Omron CX-Programmer project NewProject (CX-Programmer 9.75)

# PLC NewPLC1: CJ1M CPU11

## Global symbols (name address type ; comment)
20.00 BOOL  ; Start & Reset
20.01 BOOL  ; Kiln Consent
20.02 BOOL  ; Power OK
20.03 BOOL  ; Manual/Automatic Selector
20.04 BOOL  ; FT Enter Kiln
20.06 BOOL  ; FT Before Barrier
20.07 BOOL  ; FT Row Complete in Belts
20.08 BOOL  ; FT Row In Position
20.09 BOOL  ; FT Step-to-Step
20.10 BOOL  ; Belt Up Sensor
20.11 BOOL  ; Belt Down Sensor
20.12 BOOL  ; FT Wide Largest Row
20.13 BOOL  ; Spare
20.14 BOOL  ; Spare
20.15 BOOL  ; Spare
21.00 BOOL  ; Manual Up/Down Up
21.01 BOOL  ; Manual Up/Down Down
21.02 BOOL  ; Manual Step-To-Step Belts
21.03 BOOL  ; Manual Rollers Under Belts
21.04 BOOL  ; Manual Roller Before Barrier
21.05 BOOL  ; Manual Roller After Barrier
21.06 BOOL  ; Manual Barier Up/Down
21.07 BOOL  ; Manual Prepare Row Valve
21.08 BOOL  ; Spare
21.09 BOOL  ; Spare
21.10 BOOL  ; Spare
21.11 BOOL  ; Spare
21.12 BOOL  ; Spare
21.13 BOOL  ; Spare
21.14 BOOL  ; Spare
21.15 BOOL  ; Spare
30.00 BOOL  ; Enter Kiln Roller
30.01 BOOL  ; Barrier Valve
30.02 BOOL  ; Roller Under Barrier
30.03 BOOL  ; Roller Under Belts
30.04 BOOL  ; Up/Down Belts
30.05 BOOL  ; Up/Down Valve
30.06 BOOL  ; Preapare Row Valve
30.07 BOOL  ; Automatic Run Lamp
30.08 BOOL  ; Spare
30.09 BOOL  ; Spare
30.10 BOOL  ; Enter Kiln Roller (Slow Speed)
30.11 BOOL  ; Roller Under Barrier (Slow Speed)
30.12 BOOL  ; Sarin
30.13 BOOL  ; Sarin
30.14 BOOL  ; Unloaing Machine Consent
30.15 BOOL  ; Unloaing Machine Consent
40.00 BOOL  ; Automatic In progress
40.01 BOOL  ; Automatic Run OK
41.00 BOOL  ; Start Sequence
42.00 BOOL  ; OK Run EnterKiln Rollers
43.00 BOOL  ; Ok Run Roller Under Barrier
50.00 BOOL  ; Existence Alarm
60 CHANNEL  ; Alarms Word
70.00 BOOL  ; Start Sarin
C0001 BOOL  ; Start Fast Speed Enter Kiln Rollers Time
C0002 BOOL  ; Time Slow Speed Roller Under Barrier
C0003 BOOL  ; Stay Barrier Down Down
D100 CHANNEL  ; Start Fast Speed Enter Kiln Rollers Time
D101 CHANNEL  ; Data Time Slow Speed Roller Under Barrier
D102 CHANNEL  ; Time Barrier Stay Down
T0000 BOOL  ; Time Sarin In Start
T0001 BOOL  ; Time FT Enter Kiln Engage
T0002 BOOL  ; Time FT Enter Kiln Disengage
T0003 BOOL  ; FT Large Row Engage
T0004 BOOL  ; FT Large Row Disengage
T0005 BOOL  ; Time Restart Enter Kiln Roller
T0006 BOOL  ; Time FT Befor Brrier Engage
T0007 BOOL  ; Time FT Befor Brrier Disengage
W10.00 BOOL  ; Barrier Valve Up
W11.00 BOOL  ; Up Barrier
W11.01 BOOL  ; Down Barrier

## Program NewProgram1 (cyclic task 0)
; This Program Designed By Eng: Mahmoud Shaban Ahmed

### Section Inputs

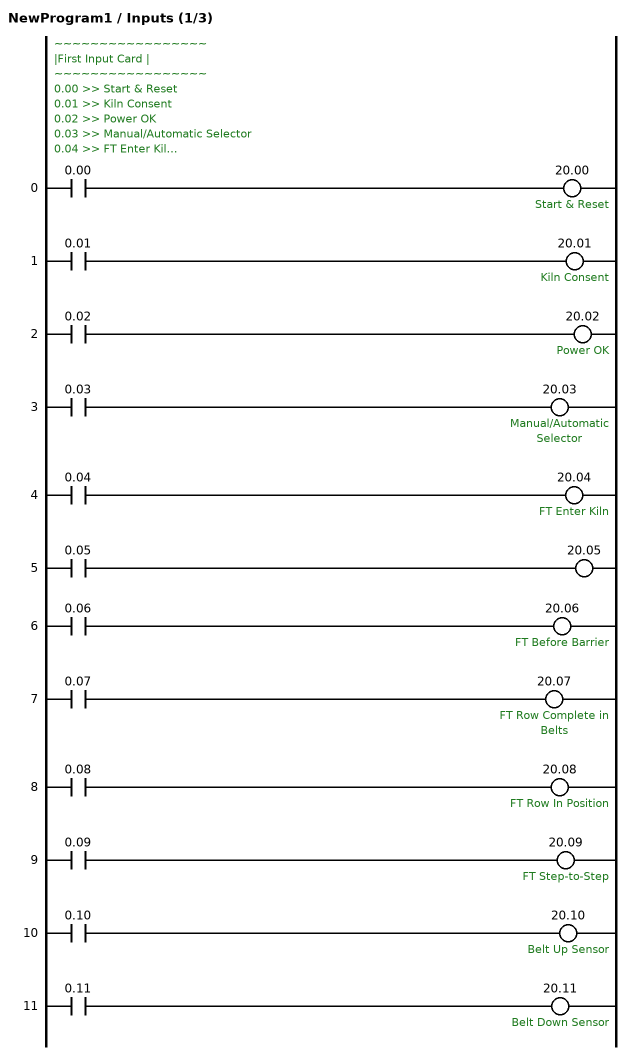
; rung 0: ~~~~~~~~~~~~~~~~~ / |First Input Card | / ~~~~~~~~~~~~~~~~~ / 0.00 >> Start & Reset / 0.01 >> Kiln Consent / 0.02 >> Power OK / 0.03 >> Manual/Automatic Selector / 0.04 >> FT Enter Kiln / 0.05 >> / 0.06 >> FT Before Barrier / 0.07 >> FT Row Complete in Belts / 0.08 >> FT Row In Position / 0.09 >> FT Step-to-Step / 0.10 >> Belt Up Sensor / 0.11 >> Belt Down Sensor / 0.12 >> FT Wide Largest Row / 0.13 >>Spare / 0.14 >>Spare / 0.15 >>Spare / >>>>>>>>>>>>>>>>>>>>>>>>>>>>>>>>>>>>>>>>>>>>>>>>>>>>>>>>>>>>>>>>>>>>>>>>>>>>>>>>>>>>>>>>>>>>>>>>>>>>>>>>>>>>>>>
LD 0.00
OUT 20.00  ; Start & Reset
; rung 1
LD 0.01
OUT 20.01  ; Kiln Consent
; rung 2
LD 0.02
OUT 20.02  ; Power OK
; rung 3
LD 0.03
OUT 20.03  ; Manual/Automatic Selector
; rung 4
LD 0.04
OUT 20.04  ; FT Enter Kiln
; rung 5
LD 0.05
OUT 20.05
; rung 6
LD 0.06
OUT 20.06  ; FT Before Barrier
; rung 7
LD 0.07
OUT 20.07  ; FT Row Complete in Belts
; rung 8
LD 0.08
OUT 20.08  ; FT Row In Position
; rung 9
LD 0.09
OUT 20.09  ; FT Step-to-Step
; rung 10
LD 0.10
OUT 20.10  ; Belt Up Sensor
; rung 11
LD 0.11
OUT 20.11  ; Belt Down Sensor

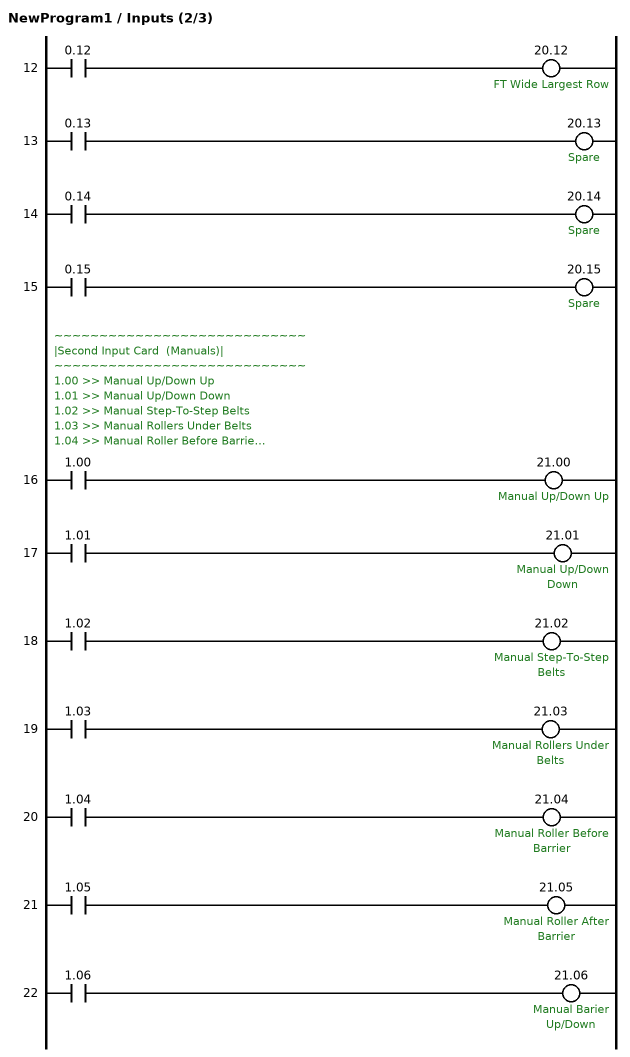
; rung 12
LD 0.12
OUT 20.12  ; FT Wide Largest Row
; rung 13
LD 0.13
OUT 20.13  ; Spare
; rung 14
LD 0.14
OUT 20.14  ; Spare
; rung 15
LD 0.15
OUT 20.15  ; Spare
; rung 16: ~~~~~~~~~~~~~~~~~~~~~~~~~~~~ / |Second Input Card  (Manuals)| / ~~~~~~~~~~~~~~~~~~~~~~~~~~~~ / 1.00 >> Manual Up/Down Up / 1.01 >> Manual Up/Down Down / 1.02 >> Manual Step-To-Step Belts / 1.03 >> Manual Rollers Under Belts / 1.04 >> Manual Roller Before Barrier / 1.05 >> Manual Roller After Barrier / 1.06 >> Manual Barier Up/Down / 1.07 >> Manual Prepare Row Valve / 1.08 >> Spare / 1.09 >> Spare / 1.10 >> Spare / 1.11 >> Spare / 1.12 >> Spare / 1.13 >> Spare / 1.14 >> Spare / 1.15 >> Spare / >>>>>>>>>>>>>>>>>>>>>>>>>>>>>>>>>>>>>>>>>>>>>>>>>>>>>>>>>>>>>>>>>>>>>>>>>>>>>>>>>>>>>>>>>>>>>>>>>>>>>>>>>>>>>>>
LD 1.00
OUT 21.00  ; Manual Up/Down Up
; rung 17
LD 1.01
OUT 21.01  ; Manual Up/Down Down
; rung 18
LD 1.02
OUT 21.02  ; Manual Step-To-Step Belts
; rung 19
LD 1.03
OUT 21.03  ; Manual Rollers Under Belts
; rung 20
LD 1.04
OUT 21.04  ; Manual Roller Before Barrier
; rung 21
LD 1.05
OUT 21.05  ; Manual Roller After Barrier
; rung 22
LD 1.06
OUT 21.06  ; Manual Barier Up/Down

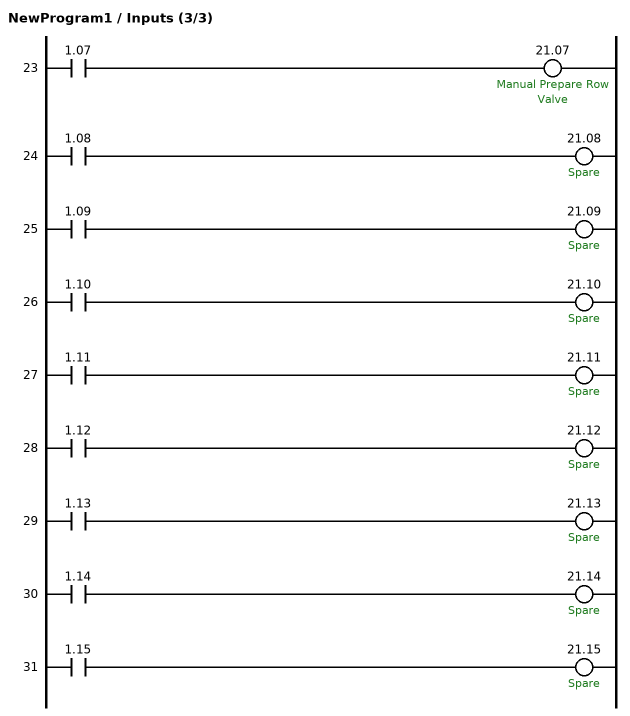
; rung 23
LD 1.07
OUT 21.07  ; Manual Prepare Row Valve
; rung 24
LD 1.08
OUT 21.08  ; Spare
; rung 25
LD 1.09
OUT 21.09  ; Spare
; rung 26
LD 1.10
OUT 21.10  ; Spare
; rung 27
LD 1.11
OUT 21.11  ; Spare
; rung 28
LD 1.12
OUT 21.12  ; Spare
; rung 29
LD 1.13
OUT 21.13  ; Spare
; rung 30
LD 1.14
OUT 21.14  ; Spare
; rung 31
LD 1.15
OUT 21.15  ; Spare

### Section Main

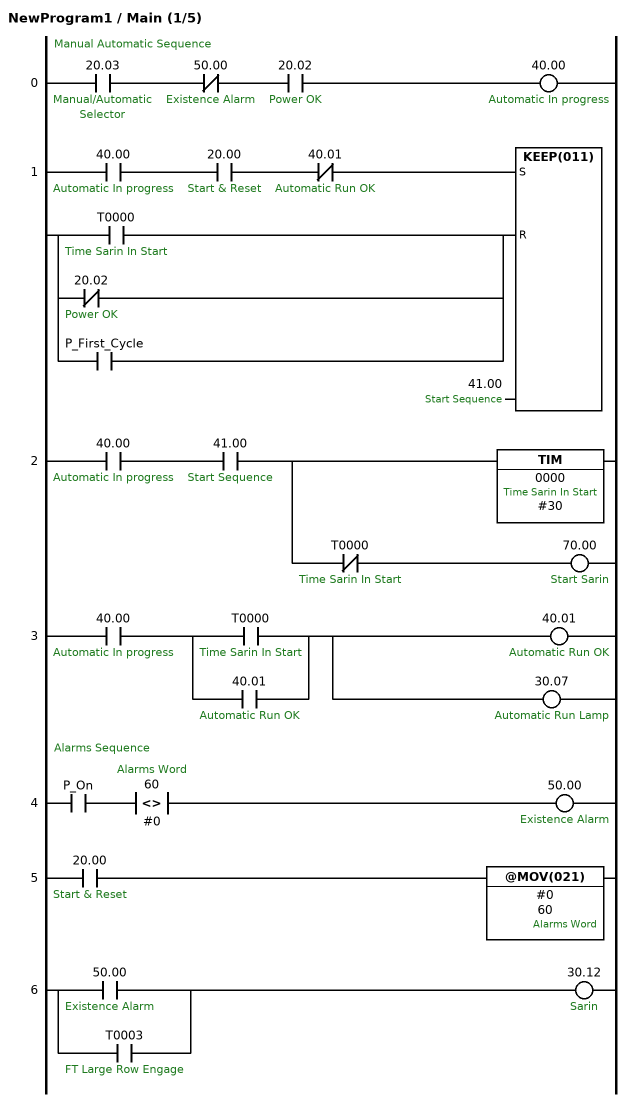
; rung 0: Manual Automatic Sequence
LD 20.03  ; Manual/Automatic Selector
ANDNOT 50.00  ; Existence Alarm
AND 20.02  ; Power OK
OUT 40.00  ; Automatic In progress
; rung 1
LD 40.00  ; Automatic In progress
AND 20.00  ; Start & Reset
ANDNOT 40.01  ; Automatic Run OK
LD T0000  ; Time Sarin In Start
ORNOT 20.02  ; Power OK
OR P_First_Cycle
KEEP(011) 41.00  ; Start Sequence
; rung 2
LD 40.00  ; Automatic In progress
AND 41.00  ; Start Sequence
TIM 0000 #30  ; Time Sarin In Start
ANDNOT T0000  ; Time Sarin In Start
OUT 70.00  ; Start Sarin
; rung 3
LD 40.00  ; Automatic In progress
LD T0000  ; Time Sarin In Start
OR 40.01  ; Automatic Run OK
ANDLD
OUT 40.01  ; Automatic Run OK
OUT 30.07  ; Automatic Run Lamp
; rung 4: Alarms Sequence
LD P_On
AND<>(305) 60 #0  ; Alarms Word
OUT 50.00  ; Existence Alarm
; rung 5
LD 20.00  ; Start & Reset
@MOV(021) #0 60  ; Alarms Word
; rung 6
LD 50.00  ; Existence Alarm
OR T0003  ; FT Large Row Engage
OUT 30.12  ; Sarin

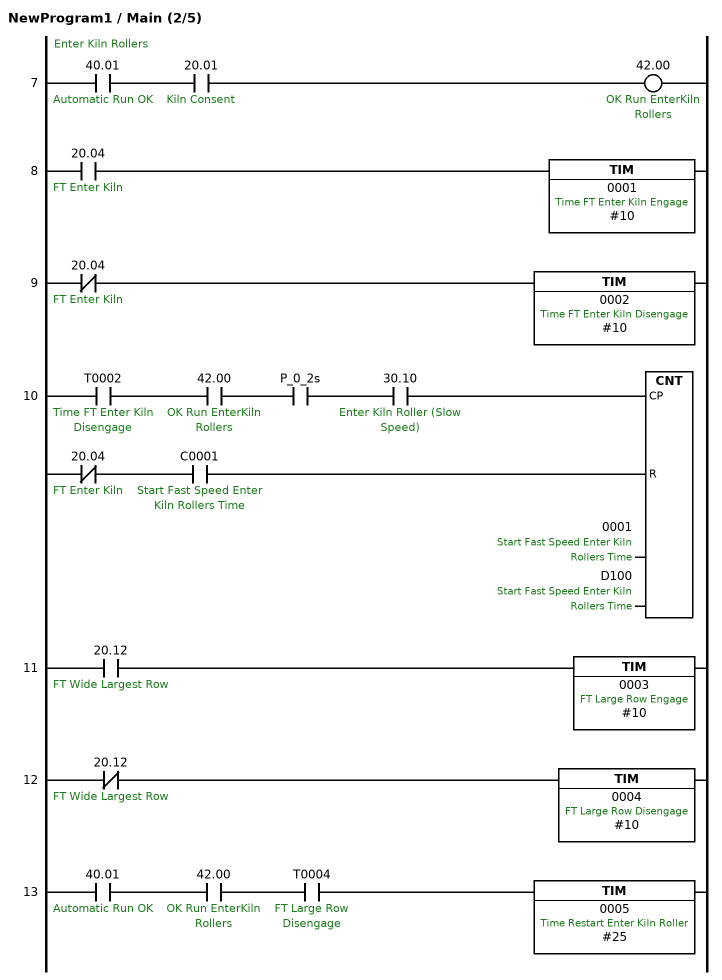
; rung 7: Enter Kiln Rollers
LD 40.01  ; Automatic Run OK
AND 20.01  ; Kiln Consent
OUT 42.00  ; OK Run EnterKiln Rollers
; rung 8
LD 20.04  ; FT Enter Kiln
TIM 0001 #10  ; Time FT Enter Kiln Engage
; rung 9
LDNOT 20.04  ; FT Enter Kiln
TIM 0002 #10  ; Time FT Enter Kiln Disengage
; rung 10
LD T0002  ; Time FT Enter Kiln Disengage
AND 42.00  ; OK Run EnterKiln Rollers
AND P_0_2s
AND 30.10  ; Enter Kiln Roller (Slow Speed)
LDNOT 20.04  ; FT Enter Kiln
AND C0001  ; Start Fast Speed Enter Kiln Rollers Time
CNT 0001 D100  ; Start Fast Speed Enter Kiln Rollers Time
; rung 11
LD 20.12  ; FT Wide Largest Row
TIM 0003 #10  ; FT Large Row Engage
; rung 12
LDNOT 20.12  ; FT Wide Largest Row
TIM 0004 #10  ; FT Large Row Disengage
; rung 13
LD 40.01  ; Automatic Run OK
AND 42.00  ; OK Run EnterKiln Rollers
AND T0004  ; FT Large Row Disengage
TIM 0005 #25  ; Time Restart Enter Kiln Roller

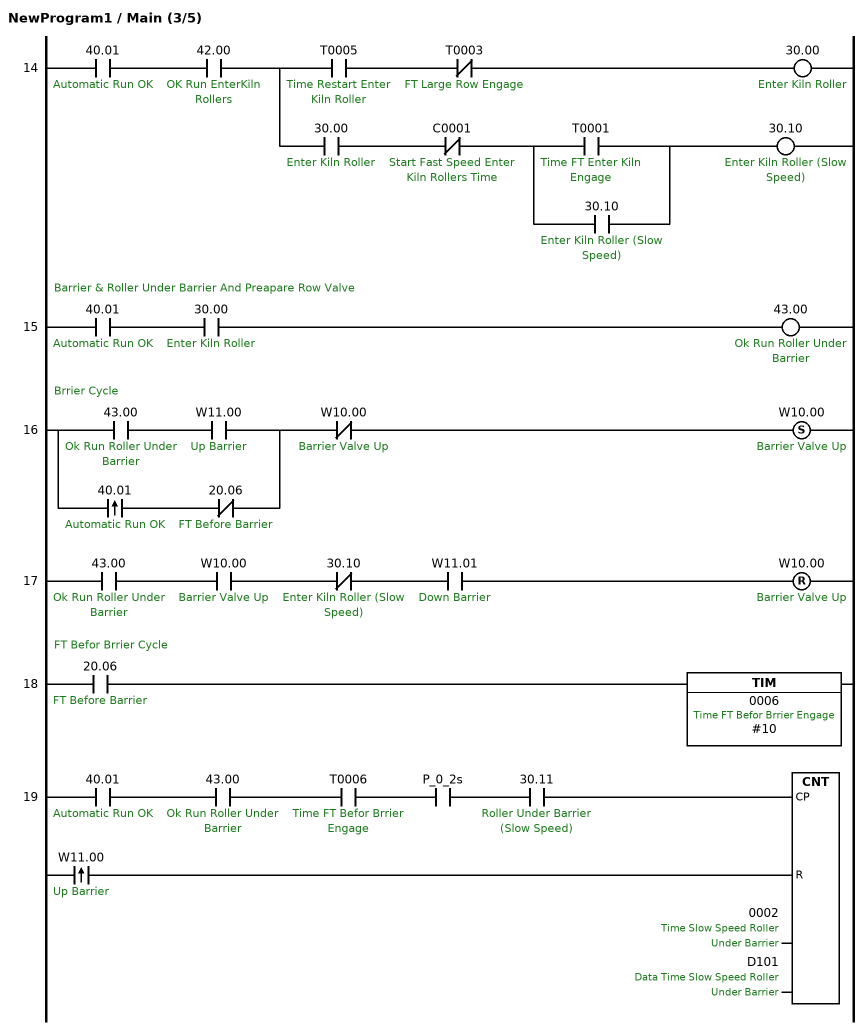
; rung 14
LD 40.01  ; Automatic Run OK
AND 42.00  ; OK Run EnterKiln Rollers
OUT TR0
AND T0005  ; Time Restart Enter Kiln Roller
ANDNOT T0003  ; FT Large Row Engage
OUT 30.00  ; Enter Kiln Roller
LD TR0
AND 30.00  ; Enter Kiln Roller
ANDNOT C0001  ; Start Fast Speed Enter Kiln Rollers Time
LD T0001  ; Time FT Enter Kiln Engage
OR 30.10  ; Enter Kiln Roller (Slow Speed)
ANDLD
OUT 30.10  ; Enter Kiln Roller (Slow Speed)
; rung 15: Barrier & Roller Under Barrier And Preapare Row Valve
LD 40.01  ; Automatic Run OK
AND 30.00  ; Enter Kiln Roller
OUT 43.00  ; Ok Run Roller Under Barrier
; rung 16: Brrier Cycle
LD 43.00  ; Ok Run Roller Under Barrier
AND W11.00  ; Up Barrier
@LD 40.01  ; Automatic Run OK
ANDNOT 20.06  ; FT Before Barrier
ORLD
ANDNOT W10.00  ; Barrier Valve Up
SET W10.00  ; Barrier Valve Up
; rung 17
LD 43.00  ; Ok Run Roller Under Barrier
AND W10.00  ; Barrier Valve Up
ANDNOT 30.10  ; Enter Kiln Roller (Slow Speed)
AND W11.01  ; Down Barrier
RSET W10.00  ; Barrier Valve Up
; rung 18: FT Befor Brrier Cycle
LD 20.06  ; FT Before Barrier
TIM 0006 #10  ; Time FT Befor Brrier Engage
; rung 19
LD 40.01  ; Automatic Run OK
AND 43.00  ; Ok Run Roller Under Barrier
AND T0006  ; Time FT Befor Brrier Engage
AND P_0_2s
AND 30.11  ; Roller Under Barrier (Slow Speed)
@LD W11.00  ; Up Barrier
CNT 0002 D101  ; Data Time Slow Speed Roller Under Barrier, Time Slow Speed Roller Under Barrier

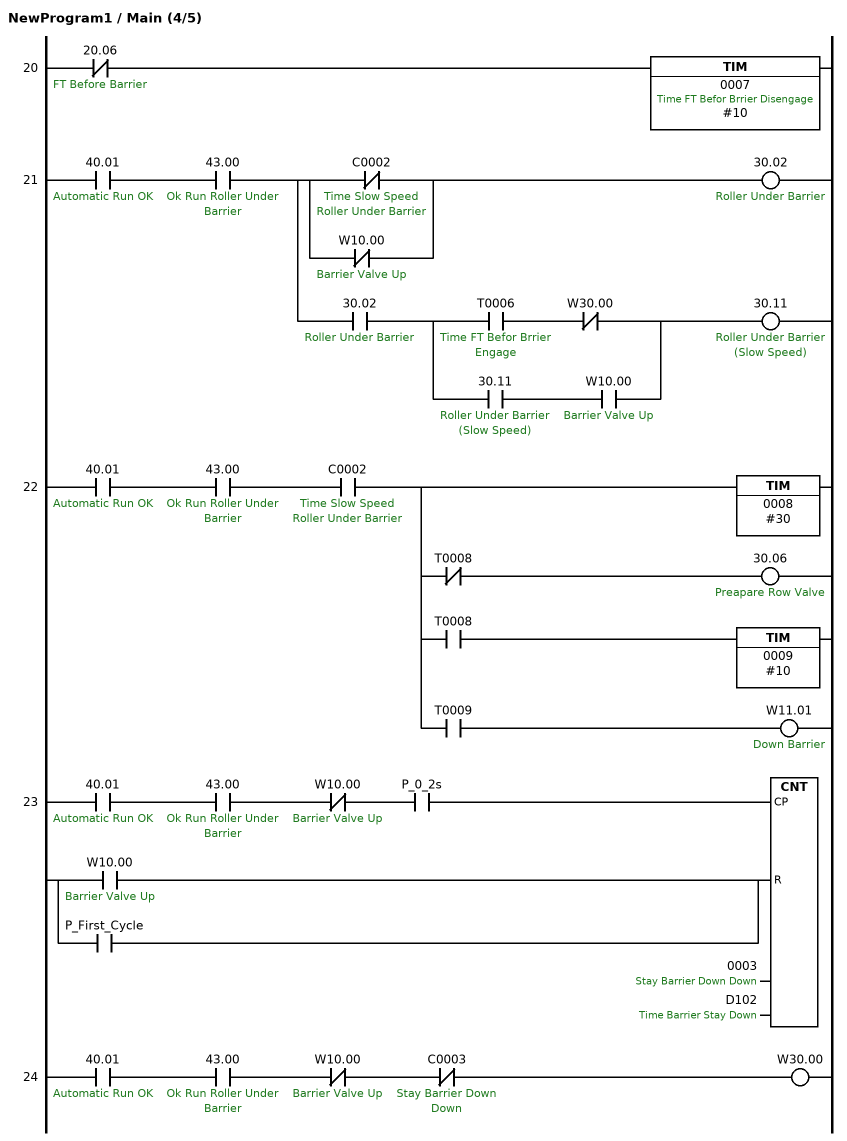
; rung 20
LDNOT 20.06  ; FT Before Barrier
TIM 0007 #10  ; Time FT Befor Brrier Disengage
; rung 21
LD 40.01  ; Automatic Run OK
AND 43.00  ; Ok Run Roller Under Barrier
OUT TR0
LDNOT C0002  ; Time Slow Speed Roller Under Barrier
ORNOT W10.00  ; Barrier Valve Up
ANDLD
OUT 30.02  ; Roller Under Barrier
LD TR0
AND 30.02  ; Roller Under Barrier
LD T0006  ; Time FT Befor Brrier Engage
ANDNOT W30.00
LD 30.11  ; Roller Under Barrier (Slow Speed)
AND W10.00  ; Barrier Valve Up
ORLD
ANDLD
OUT 30.11  ; Roller Under Barrier (Slow Speed)
; rung 22
LD 40.01  ; Automatic Run OK
AND 43.00  ; Ok Run Roller Under Barrier
AND C0002  ; Time Slow Speed Roller Under Barrier
OUT TR0
TIM 0008 #30
ANDNOT T0008
OUT 30.06  ; Preapare Row Valve
LD TR0
AND T0008
TIM 0009 #10
LD TR0
AND T0009
OUT W11.01  ; Down Barrier
; rung 23
LD 40.01  ; Automatic Run OK
AND 43.00  ; Ok Run Roller Under Barrier
ANDNOT W10.00  ; Barrier Valve Up
AND P_0_2s
LD W10.00  ; Barrier Valve Up
OR P_First_Cycle
CNT 0003 D102  ; Time Barrier Stay Down, Stay Barrier Down Down
; rung 24
LD 40.01  ; Automatic Run OK
AND 43.00  ; Ok Run Roller Under Barrier
ANDNOT W10.00  ; Barrier Valve Up
ANDNOT C0003  ; Stay Barrier Down Down
OUT W30.00

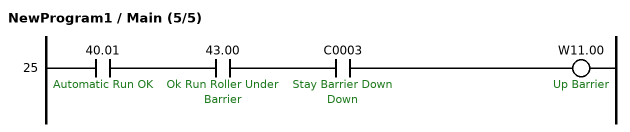
; rung 25
LD 40.01  ; Automatic Run OK
AND 43.00  ; Ok Run Roller Under Barrier
AND C0003  ; Stay Barrier Down Down
OUT W11.00  ; Up Barrier

### Section OutPuts

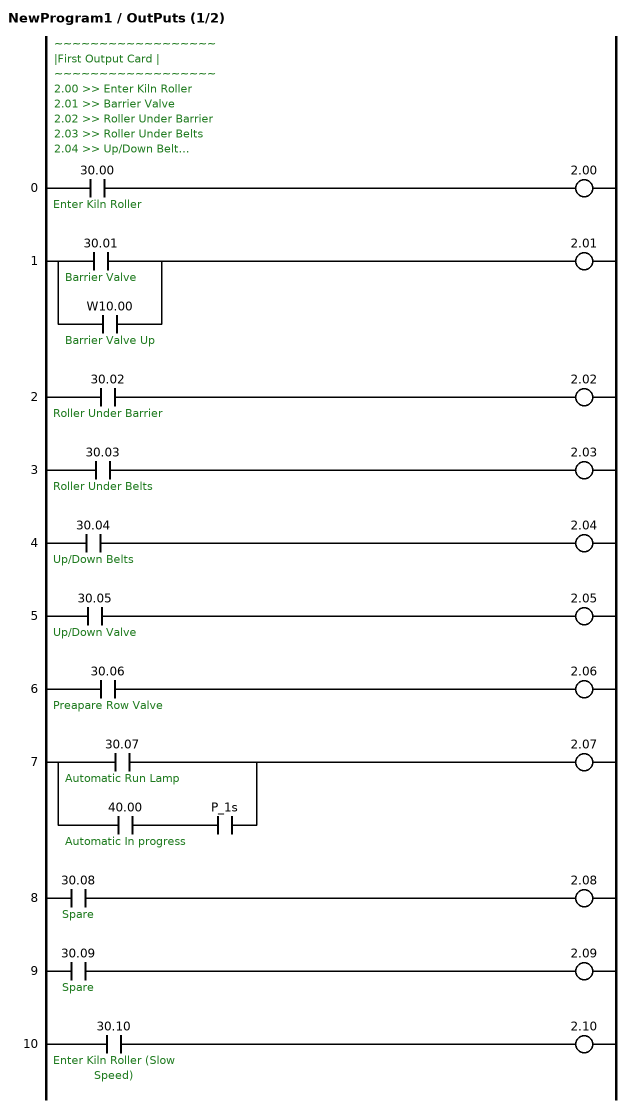
; rung 0: ~~~~~~~~~~~~~~~~~~ / |First Output Card | / ~~~~~~~~~~~~~~~~~~ / 2.00 >> Enter Kiln Roller / 2.01 >> Barrier Valve / 2.02 >> Roller Under Barrier / 2.03 >> Roller Under Belts / 2.04 >> Up/Down Belts / 2.05 >> Up/Down Valve / 2.06 >> Preapare Row Valve / 2.07 >> Automatic Run Lamp / 2.08 >> Spare / 2.09 >> Spare / 2.10 >> Enter Kiln Roller (Slow Speed) / 2.11 >> Roller Under Barrier (Slow Speed) / 2.12 >> Sarin / 2.13 >> Sarin / 2.14 >> Unloaing Machine Consent / 2.15 >> Unloaing Machine Consent / >>>>>>>>>>>>>>>>>>>>>>>>>>>>>>>>>>>>>>>>>>>>>>>>>>>>>>>>>>>>>>>>>>>>>>>>>>>>>>>>>>>>>>>>>>>>>>>>>>>>>>>>>>>>>>>
LD 30.00  ; Enter Kiln Roller
OUT 2.00
; rung 1
LD 30.01  ; Barrier Valve
OR W10.00  ; Barrier Valve Up
OUT 2.01
; rung 2
LD 30.02  ; Roller Under Barrier
OUT 2.02
; rung 3
LD 30.03  ; Roller Under Belts
OUT 2.03
; rung 4
LD 30.04  ; Up/Down Belts
OUT 2.04
; rung 5
LD 30.05  ; Up/Down Valve
OUT 2.05
; rung 6
LD 30.06  ; Preapare Row Valve
OUT 2.06
; rung 7
LD 30.07  ; Automatic Run Lamp
LD 40.00  ; Automatic In progress
AND P_1s
ORLD
OUT 2.07
; rung 8
LD 30.08  ; Spare
OUT 2.08
; rung 9
LD 30.09  ; Spare
OUT 2.09
; rung 10
LD 30.10  ; Enter Kiln Roller (Slow Speed)
OUT 2.10

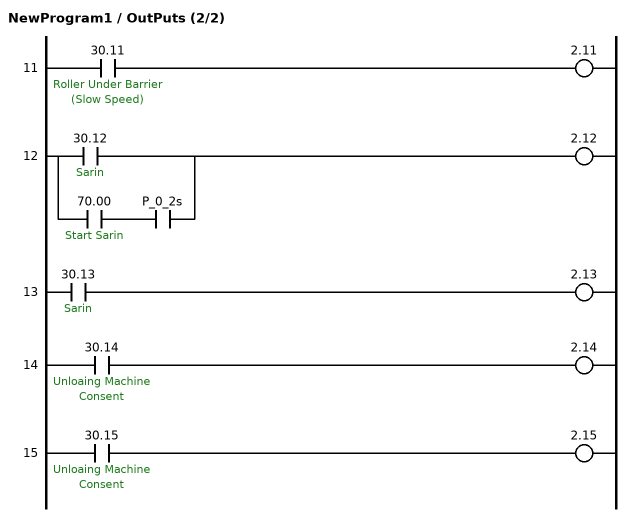
; rung 11
LD 30.11  ; Roller Under Barrier (Slow Speed)
OUT 2.11
; rung 12
LD 30.12  ; Sarin
LD 70.00  ; Start Sarin
AND P_0_2s
ORLD
OUT 2.12
; rung 13
LD 30.13  ; Sarin
OUT 2.13
; rung 14
LD 30.14  ; Unloaing Machine Consent
OUT 2.14
; rung 15
LD 30.15  ; Unloaing Machine Consent
OUT 2.15

### Section END
; rung 0
END(001)